(* Logix 5000 project; controller Lab1 vendor 1 type 14 code 155 rev 20.12; software revision 20.01 *)

TASK MainTask (continuous, watchdog 500 ms) : MainProgram

MODULES
   Local : vendor 1 type 14 code 155 (PointIO 0, rev 20.12)
      A_In : 1734-IE2V (PointIO 2, rev 3.1, Input RPI 80 ms)
      Stepper_1 : vendor 10 type 150 code 185 (PointIO 5, rev 1.1, Output RPI 50 ms)
      Stepper_2 : vendor 10 type 150 code 185 (PointIO 6, rev 1.1, Output RPI 50 ms)
      Discrete_IO : Embedded (PointIO 1, rev 20.11, Output RPI 20 ms)
      A_Out : 1734-OE2V (PointIO 3, rev 3.1, Output RPI 80 ms)
      HSC : vendor 1 type 109 code 13 (PointIO 4, rev 3.1, Output RPI 80 ms)
END_MODULES

PROGRAM MainProgram   (* main routine MainRoutine *)
VAR
   C6 : COUNTER := (PRE := 8);
   C7 : COUNTER;
   T3 : TIMER := (PRE := 5000);
   T4 : TIMER := (PRE := 5000);
   T5 : TIMER := (PRE := 5000);
   VAR1 : BOOL;
END_VAR

ROUTINE MainRoutine   (* ladder *)
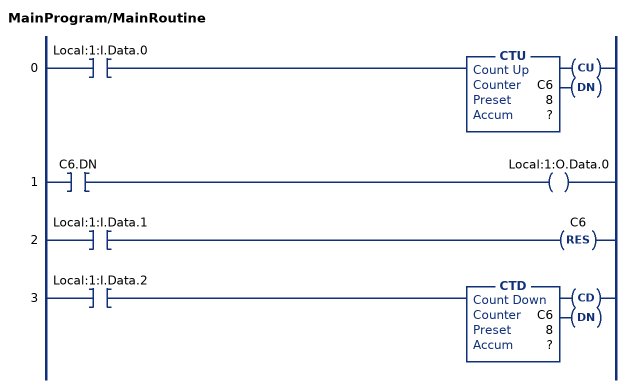
   0: XIC(Local:1:I.Data.0)CTU(C6,?,?);
   1: XIC(C6.DN)OTE(Local:1:O.Data.0);
   2: XIC(Local:1:I.Data.1)RES(C6);
   3: XIC(Local:1:I.Data.2)CTD(C6,?,?);
END_ROUTINE
END_PROGRAM
